{attribute 'GeneratedUsingTerminal: EP1816-1008-0016'}
{attribute addProperty BoxType "EP1816-1008-0016"}
{attribute addProperty Id "InputAT %I*ARRAY[0..7] OF BOOL8"}
{attribute addProperty CRC "3697175534"}
{attribute addProperty Size "8"}
TYPE DIG_Inputs_Channel_38F9DD27 :
STRUCT
	{attribute addProperty Name "Input"}
	Input AT %I* : ARRAY[0..7] OF BOOL;
END_STRUCT
END_TYPE

(* stored: Version 1.2.0.0, ProductVersion 3.1.4024.9
   DUT DIG_Inputs_Channel_38F9DD27: Id {e6b27ebf-a1ab-4712-b347-2cbe7d726f7c} *)
